Staubli VAL3: exceptionHandle.pjx

--- exceptionHandle.pjx ---
Parameters version=s7.9.1 stackSize=5000 millimeterUnit=true
Program file=exceptionForce.pgx
Program file=exceptionRobot.pgx
Program file=exceptionRos.pgx
Program file=start.pgx
Program file=stop.pgx
Data file=exceptionHandle.dtx
Type name=FlagStatus path=Disk://RobotController_Libs/FlagStatus/FlagStatus.pjx
Type name=RobotStatus path=Disk://RobotController_Libs/RobotStatus/RobotStatus.pjx

--- exceptionHandle.dtx ---
mdesc mNomSpeed
public num nForceThreshold[6]
public num nSpeedThreshold[6]
public num nRosFlagCmd

--- exceptionForce.pgx ---
public program exceptionForce(num& x_nSensorForce[], FlagStatus& x_fSensorStatus)
begin

  //This program is used for handling the exception of the interaction force/torque between the robot endeffector
  //and the operation object in the environment. When the detected force/torqure from the sensor exceeds the force/torqure
  //threshold(setted in advance), the robot should be stopped to protect itself and the operation object
  //from being damaged.

  //Firstly, the force/torque threshold of interactive operation in different main axies should be defined for safety.
  nForceThreshold[0]=5
  nForceThreshold[1]=5
  nForceThreshold[2]=5
  nForceThreshold[3]=0.2
  nForceThreshold[4]=0.2
  nForceThreshold[5]=0.2

  //Secondly, the interactive force/torque between the robot endeffector and operated object in the environment should
  //be detected and acquired from the sensor. And by comparing the detected force/torque values with set safe threshold
  //of the force/torque, the robot motion should be decided whether the robot stops moving or keeps moving.
  if x_nSensorForce<=nForceThreshold
    x_fSensorStatus.ForceFlag=1
  else
    x_fSensorStatus.ForceFlag=-1
  endIf

end

--- exceptionRobot.pgx ---
public program exceptionRobot(RobotStatus& x_rRobotStatus, FlagStatus& x_fRobotStatus)
begin

  //This program is used for checking the current robot status(motion, running) and deciding whether
  //the robot is running normally. And the robot will be stopped for safety if abnormal situation occurs
  //for the robot, otherwise the robot keeps running normally.

  //The robot will react if the abnormal situation occurs.(the robot has own safety portection mechanism)
  //Unit: m/s, degree/s
  nSpeedThreshold[0]=0.5
  nSpeedThreshold[1]=0.5
  nSpeedThreshold[2]=0.5
  nSpeedThreshold[3]=90
  nSpeedThreshold[4]=90
  nSpeedThreshold[5]=90

  if x_rRobotStatus.cartesianSpace.CartesianVel<=nSpeedThreshold
    x_fRobotStatus.RosFlag=1
  else
    x_fRobotStatus.RosFlag=-1
  endIf

end

--- exceptionRos.pgx ---
public program exceptionRos(FlagStatus& x_fRosStatus, num& x_nRosFlagCmd)
begin

  //This program is used for checking the ROS command of exception handling from the host ROS controller
  //and deciding whether the robot should keep executing the motion command or not.

  //The ROS command flag from the host ROS controller should be acquired through TCP/IP socket communication.
  //And the ROS flag in the ROS massage command is in the last element in the received array.
  x_fRosStatus.RosFlag=x_nRosFlagCmd

end
